TYPE ST_MGMT_ThNTZ_Aktor_Stellwert :
STRUCT
	Betrieb			: BOOL;
END_STRUCT
END_TYPE

(* stored: Version 1.1.0.1, ProductVersion 3.1.4024.9
   DUT ST_MGMT_ThNTZ_Aktor_Stellwert: Id {eacb48fd-ab5b-411c-a503-cfc25cdfe437} *)
